// TIA Portal V20 export
// export: Created 2026-07-10T11:12:25.6583691Z, ExportSetting WithDefaults, DisplayName Totally Integrated Automation Portal, DisplayVersion V20, DisplayName TIA Portal Openness, DisplayVersion V20, DisplayName TIA Portal Version Control Interface, DisplayVersion V20, DisplayName STEP 7 Professional, DisplayVersion V20, DisplayName STEP 7 Safety, DisplayVersion V20, DisplayName WinCC Basic/Comfort/Advanced, DisplayVersion V20, DisplayName WinCC Unified, DisplayVersion V20
FUNCTION_BLOCK "Weighting"   // FB18, SCL
{ S7_Optimized_Access := 'FALSE' }
VERSION : 0.1
// stored: AutoNumber true, IsIECCheckEnabled false, SetENOAutomatically false, UDAEnableTagReadback false
   VAR DB_SPECIFIC
      buffer1 { S7_SetPoint := 'True'} : Array[0..1] of Word;
      buffer2 : Array[0..1] of Word;
      Enable { S7_SetPoint := 'True'} : Bool;
      ManualValueProvided1 : Bool;
      ManualValueProvided2 : Bool;
      ManualValue1 : Real;
      ManualValue2 : Real;
   END_VAR
   VAR
      WeightHandlers : Array[0..1] of "WeightHandler";
      TankWeigher1 { S7_SetPoint := 'True'} : "TankWeigher";
   END_VAR
   VAR DB_SPECIFIC
      RetainData : "WeightRetainData";
      TimeNow { S7_SetPoint := 'True'} : DTL;
   END_VAR
   VAR_TEMP
      Temp1 : DWord;
      Temp2 : DWord;
      Ret : Int;
   END_VAR
   VAR CONSTANT
      CLOR_DENSITY : Real := 1.2;
   END_VAR
BEGIN
   #Enable := "MB".Table.WeightingEnable;

   "ModbusLoad"(REQ :="FirstScan",
               PORT := "Local~CM_1241_(RS422_485)_1",
               BAUD := 9600,
               PARITY := 0,
               RESP_TO := 100,
               MB_DB := "ModbusMaster");

   "ModbusMaster"(REQ := "ModbusLoad".DONE,
                 MB_ADDR := 16,
                 MODE := 0,
                 DATA_ADDR := 40063,
                 DATA_LEN := 2,
                 DATA_PTR := "MB".Table.SensorWeightVoltage1);

   "ModbusMaster"(REQ := "ModbusLoad".DONE,
                 MB_ADDR := 17,
                 MODE := 0,
                 DATA_ADDR := 40063,
                 DATA_LEN := 2,
                 DATA_PTR := "MB".Table.SensorWeightVoltage2);

   "ModbusMaster"(REQ := "ModbusLoad".DONE,
                 MB_ADDR := 18,
                 MODE := 0,
                 DATA_ADDR := 40005,
                 DATA_LEN := 2,
                 DATA_PTR := "MB".Table.WaterTemperature);


   IF NOT #Enable THEN
       IF "MB".Table.Weighting_SaveManualValue THEN
           IF "MB".Table.Weighting_ManualValue1 <> 0 THEN
               #ManualValueProvided1 := TRUE;
               #ManualValue1 := "MB".Table.Weighting_ManualValue1 * #CLOR_DENSITY;
           END_IF;
           IF "MB".Table.Weighting_ManualValue2 <> 0 THEN
               #ManualValueProvided2 := TRUE;
               #ManualValue2 := "MB".Table.Weighting_ManualValue1 * #CLOR_DENSITY;
           END_IF;
       END_IF;
   ELSE
       #ManualValueProvided1 := FALSE;
       #ManualValue1 := 0;
       #ManualValueProvided2 := FALSE;
       #ManualValue1 := 0;
   END_IF;

   IF "MB".Table.Weighting_SaveManualValue THEN
       "MB".Table.Weighting_SaveManualValue := FALSE;
   END_IF;



   #WeightHandlers[0](
                      Value := "MB".Table.SensorWeightVoltage1,
                      ValueMin := "MB".Table.WeightVoltageMin1,
                      ValueMax := "MB".Table.WeightVoltageMax1,
                      ValueOffset := "MB".Table.WeightValueOffset1,
                      OutputMin := "MB".Table.WeightValueMin1,
                      OutputMax := "MB".Table.WeightValueMax1,
                      Output => "MB".Table.WeightValue1);

   #WeightHandlers[1](
                      Value := "MB".Table.SensorWeightVoltage2,
                      ValueMin := "MB".Table.WeightVoltageMin2,
                      ValueMax := "MB".Table.WeightVoltageMax2,
                      ValueOffset := "MB".Table.WeightValueOffset2,
                      OutputMin := "MB".Table.WeightValueMin2,
                      OutputMax := "MB".Table.WeightValueMax2,
                      Output => "MB".Table.WeightValue2);

   #Ret := RD_SYS_T(#TimeNow);

   #TankWeigher1(WeightDelay:="MB".Table.WeightingDelay*1000,
                 WeightDeadZone:="MB".Table.WeightingDeadZone,
                 DayTour:="MB".Table.CycleDay,
                 CalendarMonth := #TimeNow.MONTH,
                 CalendarDay := #TimeNow.DAY,
                 ref_RetainData:=#RetainData
   );

   IF #ManualValueProvided1 THEN
       "MB".Table.WeightValue1 := #ManualValue1;
   END_IF;

   IF #ManualValueProvided2 THEN
       "MB".Table.WeightValue2 := #ManualValue2;
   END_IF;

   "MB".Table.WeightValue1Liters := "MB".Table.WeightValue1/ #CLOR_DENSITY;
   "MB".Table.WeightValue2Liters := "MB".Table.WeightValue2 / #CLOR_DENSITY;

   "MB".Table.WeightingStat_CalendarDay := #RetainData.ArrayCalendarDay;
   "MB".Table.WeightingStat_CalendarMonth := #RetainData.ArrayCalendarMonth;
   "MB".Table.WeightingStat_DayCycle := #RetainData.ArrayDayTour;
   "MB".Table.WeightingStat_Counsumed1 := #RetainData.ArrayConsumedFeed1;
   "MB".Table.WeightingStat_Load1 := #RetainData.ArrayLoadedFeed1;
   "MB".Table.WeightingStat_Counsumed2 := #RetainData.ArrayConsumedFeed2;
   "MB".Table.WeightingStat_Load2 := #RetainData.ArrayLoadedFeed2;
   "MB".Table.WeightSensor1Error := #WeightHandlers[0].Error;
   "MB".Table.WeightSensor2Error := #WeightHandlers[1].Error;
END_FUNCTION_BLOCK
